FUNCTION_BLOCK FB_Axes
VAR_INPUT
	AxesPosition:INT;
	Extended:BOOL;
	Axes_Step:Int:=0;
END_VAR
VAR
END_VAR

END_FUNCTION_BLOCK

(* stored: Version 1.1.0.1, ProductVersion 3.1.4024.3
   POU FB_Axes: Id {9a888a9c-6387-480b-81ff-ad6e9015ae81}, SpecialFunc None *)
